FUNCTION Tick : BOOL
VAR_INPUT
	nTimeInMs	: ULINT;
	nTaskInMs	: ULINT := 20;
END_VAR

Tick := (GetUnixTime() MOD (nTimeInMs * 10_000)) < (nTaskInMs * 10_000);

END_FUNCTION

(* stored: Version 1.1.0.1
   POU Tick: Id {af0eb983-e1a9-488e-9880-a3e02be9a6ad}, SpecialFunc None *)
